{attribute 'Tc2GvlVarNames'}
{attribute 'strict'}
(* Identifica lo stato della Lettura del BC:	0= Non Ancora letto/Da Leggere *)
TYPE e_Stato_LetturaBarCode :
(
	LETTURA_BC_NON_EFFETTUATA 	:= 0, // BARCODE Non Ancora letto/Da Leggere	
	LETTURA_BC_IN_CORSO			:= 1, // Lettura BARCODE In corso
	LETURA_BC_TERMINATA			:= 2, // Codice BARCODE Letto e Valido/Non da leggere, 
	LETTURA_BC_ERRATA			:= 3  // Errore durante la lettura del BARCODE 
);
END_TYPE

(* stored: Version 1.1.0.1, ProductVersion 3.1.4024.11
   EnumerationTextList e_Stato_LetturaBarCode: Id {d680159e-c965-4b54-834c-f88573c7ac5d} *)
